{attribute addProperty BoxType "AX5191-0000-0212-0212"}
{attribute addProperty Id "AdsAddrAT %I*AMSADDR6480DcOutputShiftAT %I*DINT3240DcInputShiftAT %I*DINT3240Chn0AT %I*USINT810StateAT %I*UINT1620"}
{attribute addProperty CRC "2930868045"}
{attribute addProperty SizeInBites "152"}
{attribute addProperty SizeInBytes "19"}
TYPE InfoData_AEB17F4D :
STRUCT
	{attribute addProperty Name "AdsAddr"}
	AdsAddr AT %I* : AMSADDR;
	{attribute addProperty Name "DcOutputShift"}
	DcOutputShift AT %I* : DINT;
	{attribute addProperty Name "DcInputShift"}
	DcInputShift AT %I* : DINT;
	{attribute addProperty Name "Chn0"}
	Chn0 AT %I* : USINT;
	{attribute addProperty Name "State"}
	State AT %I* : UINT;
END_STRUCT
END_TYPE

(* stored: Version 1.2.0.0, ProductVersion 3.1.4024.9
   DUT InfoData_AEB17F4D: Id {137868d0-cae0-4600-91bb-8865cc4b214e} *)
